// Mitsubishi GX Works2 project: questão_5   PLC: Q03UDV
// LRI_2023

PROGRAM MAIN
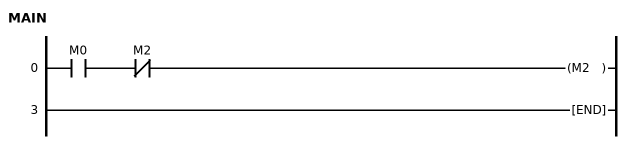
0     LD      M0
      ANI     M2
      OUT     M2
3     END
END_PROGRAM
